TYPE ST_FingerprintKey :
STRUCT
	MachineId		: 	STRING(49);//指纹器编号	
	UserId			:	STRING(49);//用户名	
	UserClassLevel	: 	STRING(49);//用户权限	
	Fid				: 	STRING(49);//本地文件id	
	MatchScore		:	STRING(49);//指纹匹配评分	
	Result			: 	STRING(49);//匹配结果	
	FileName		: 	STRING(49);//本地文件路径	
END_STRUCT
END_TYPE

(* stored: Version 1.1.0.1, ProductVersion 3.1.4024.12
   DUT ST_FingerprintKey: Id {b89b347e-189d-4b67-b372-133f617f3128} *)
